(* CODESYS project PLC_PRG.export

Project tree, tasks and I/O mapping:
  program PLC_PRG [ST]: ACT_MQTT_PUBLISHER
*)

// PLC_PRG
PROGRAM PLC_PRG
VAR
	MQTT_CLIENT : MQTT.MQTTClient;
	MQTT_PUBISHER : MQTT.MQTTPublish;
	MQTT_SUBSCRIBER : MQTT.MQTTSubscribe;
	// MQTT Client
	xEnable : BOOL;
	wsUsername : WSTRING;
	wsPassword : WSTRING;
	uiPort : UINT := 1883;
	sHostname : STRING := 'broker.hivemq.com';
	
	// MQTT Publisher
	xPublish : BOOL;
	sPayload : STRING := '{"Data": 30}';
	udiPayloadSize : UDINT ;
	wsTopic : WSTRING(1024) := "MqttTester";
	
	// MQTT Subscriber
	xSubscribe : BOOL;
	sPayloadSub : STRING;
	udiPayloadSizeSub : UDINT ;	
	wsTopicSub : WSTRING(1024);
	
	// MAIN ROUTINE
	iPublisher : INT := 1;
	xStart : BOOL;
	iValue : INT := 2;
	delay : TON;
	
END_VAR

ACT_MQTT_PUBLISHER();

udiPayloadSize := INT_TO_UDINT(LEN(sPayload));
udiPayloadSizeSub := SIZEOF(sPayloadSub);

// Delay timer
delay(IN:=, PT:= T#3S, Q=>);
// Publisher routine
CASE iPublisher OF 
	1:
	IF xStart THEN
		// Enable client
		xEnable := TRUE;
		
		IF MQTT_CLIENT.xConnectedToBroker THEN
			iPublisher := 2;
		END_IF
		
	END_IF
	2:
	IF MQTT_CLIENT.xConnectedToBroker THEN
		// set message {"Data": 20}
		sPayload := concat('{"Data":', concat(INT_TO_STRING(iValue),'}'));
		// publish message
		xPublish := TRUE;
		delay.IN := TRUE;
		iPublisher := 3;
	END_IF
	3:
	IF delay.Q AND MQTT_PUBISHER.xDone THEN
		delay.IN := FALSE;
		iValue := iValue +5;
		xPublish := FALSE;
		iPublisher := 2;
	END_IF
	
END_CASE

ACTION ACT_MQTT_PUBLISHER:
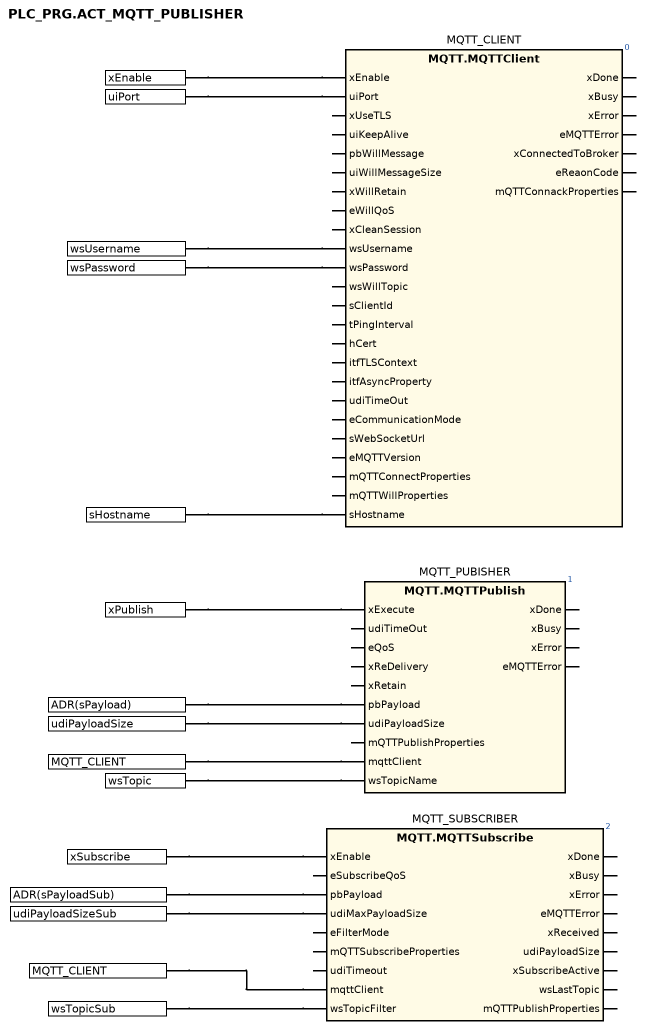
MQTT_CLIENT(
    xEnable := xEnable,
    uiPort := uiPort,
    wsUsername := wsUsername,
    wsPassword := wsPassword,
    sHostname := sHostname); // MQTT.MQTTClient
MQTT_PUBISHER(
    xExecute := xPublish,
    pbPayload := ADR(sPayload),
    udiPayloadSize := udiPayloadSize,
    mqttClient := MQTT_CLIENT,
    wsTopicName := wsTopic); // MQTT.MQTTPublish
MQTT_SUBSCRIBER(
    xEnable := xSubscribe,
    pbPayload := ADR(sPayloadSub),
    udiMaxPayloadSize := udiPayloadSizeSub,
    mqttClient := MQTT_CLIENT,
    wsTopicFilter := wsTopicSub); // MQTT.MQTTSubscribe
END_ACTION

END_PROGRAM
